TYPE EtcSlaveBase_82538BE2 :
STRUCT
END_STRUCT
END_TYPE

(* stored: Version 1.2.0.0, ProductVersion 3.1.4024.11
   DUT EtcSlaveBase_82538BE2: Id {7271e4bc-6cd0-4045-8033-11a3c83c540a} *)
